{attribute 'linkalways'} 
{attribute 'no_explicit_call' := 'This FB is a CLASS and must be accessed using methods or properties'}
{attribute 'enable_dynamic_creation'}
FUNCTION_BLOCK Node_F_VN_ConvertElementTypeExp EXTENDS VisionNode
VAR
    ipSrcImage : _ITcVnImage;
    ipDestImage : _ITcVnImage;
    eElementType : _ETcVnElementType(ETcVnElementType.TCVN_ET_SAME_AS_SOURCE);
    fScaleFactor : _LREAL(0.0);
    fDelta : _LREAL(0.0);
    hrPrev : _HRESULT(S_OK);
	hresult : _HRESULT(S_OK);
END_VAR

METHOD PUBLIC  Clone : I_Node
VAR
	pNode : POINTER TO Node_F_VN_ConvertElementTypeExp;
END_VAR
pNode := __NEW(Node_F_VN_ConvertElementTypeExp);
Clone := pNode^;
END_METHOD

METHOD FB_init : BOOL
VAR_INPUT
	bInitRetains : BOOL; // if TRUE, the retain variables are initialized (warm start / cold start)
	bInCopyCode : BOOL;  // if TRUE, the instance afterwards gets moved into the copy code (online change)
END_VAR
AddInput('ipSrcImage', ipSrcImage);
AddInput('hrPrev', hrPrev);
AddParameter('eElementType', eElementType);
AddParameter('fScaleFactor', fScaleFactor);
AddParameter('fDelta', fDelta);
AddOutput('ipDestImage', ipDestImage);
AddOutput('hresult',hresult);
END_METHOD

METHOD PROTECTED OnExecute : HRESULT
hresult.Value := F_VN_ConvertElementTypeExp(
    ipSrcImage := ipSrcImage.Value,
	ipDestImage := ipDestImage.Value,
    eElementType := eElementType.Value,
    fScaleFactor := fScaleFactor.Value,
    fDelta := fDelta.Value,
	hrPrev:= hrPrev.Value);
END_METHOD

METHOD PUBLIC PreExecutionCheck
VAR_INPUT
	Check : I_PreExecutionChecks;
END_VAR
IF FAILED(hrPrev.Value) THEN
    RETURN;
END_IF

Check.IsTrue(ipSrcImage.IsValid, 'ipSrcImage must contain an image');
END_METHOD

END_FUNCTION_BLOCK

(* stored: Version 1.1.0.1, ProductVersion 3.1.4024.13
   POU Node_F_VN_ConvertElementTypeExp: Id {04d07ce4-6f16-0b1f-0e56-e1d76b8cc0ce}, SpecialFunc None
   Folder Constructor: Id {620ff536-45ba-0311-1167-c5d9ad9db917}
   Method Clone: Id {c6dd9fd8-6586-0268-2deb-7def636c750f}
   Method FB_init: Id {f0897bbc-8b7c-088b-06e7-9648b9f7cf07}
   Method OnExecute: Id {96549d2d-7836-0c52-3b6b-0321b40e7267}
   Method PreExecutionCheck: Id {55e1f524-6563-0d2e-3ce1-fa5aeca4315c} *)
